FUNCTION_BLOCK FB_SimMotor
VAR_IN_OUT
	stMotionStage: DUT_MotionStage;
END_VAR
VAR
	fbMotionStage: FB_MotionStage;
END_VAR

stMotionStage.bLimitBackwardEnable := TRUE;
stMotionStage.bLimitForwardEnable := TRUE;
stMotionStage.bHardwareEnable := TRUE;
stMotionStage.bPowerSelf := TRUE;
stMotionStage.nEnableMode := ENUM_StageEnableMode.STAGE_ENABLE_ALWAYS;
fbMotionStage(stMotionStage := stMotionStage);

END_FUNCTION_BLOCK

(* stored: Version 1.1.0.1, ProductVersion 3.1.4022.12
   POU FB_SimMotor: Id {95f2573d-9f2a-46cf-9236-6b3c25d058e1}, SpecialFunc None *)
